(* PLC project Tc2_Utilities.FB_CalcHashValue.update Demo, tc3-libraries-kb TwinCAT 3.1 *)
(* stored: creationDateTime 2026-05-11T00:00:00, modificationDateTime 2026-05-11T00:00:00 *)

PROGRAM P_Demo_FB_CalcHashValue_update
  VAR
    fbCalc : FB_CalcHashValue;  (* Tc2_Utilities.FB_CalcHashValue 实例 *)
    eMode : E_HashMode := E_HashMode.HashMode_Sha512;  (* Hash 模式 *)
    sInput : STRING := 'hello';  (* 输入字符串 *)
    bStart : BOOL;  (* start() 返回值 *)
    bUpdate : BOOL;  (* update() 返回值 *)
  END_VAR

            // ============================================================
// Tc2_Utilities.FB_CalcHashValue.update() 演示程序（METHOD）
// ============================================================
// 验证步骤：
//   1. 引用 Tc2_Utilities
//   2. 编译 + 登录
//   3. 在线写值 sInput，观察 bStart 与 bUpdate
//   4. 完整流程需要紧接调用 finish()，见 FB_CalcHashValue.md
// ============================================================

// 先 start 才能 update
bStart  := fbCalc.start(hashMode := eMode);
bUpdate := fbCalc.update(pData := ADR(sInput), nData := LEN(sInput));

          
END_PROGRAM
